(* CoDeSys 2.3.9.28 project: TEST IO.pro *)
(* Libraries: Ethernet.lib 2.12.10 13:48:32, mod_com.lib 2.12.10 13:48:32, ModbusEthernet_04.lib 2.12.10 13:48:36, Standard.lib 2.12.10 13:48:34, SYSLIBCALLBACK.LIB 2.12.10 13:48:32 *)

(* PLC configuration (modules and I/O channels)
0750-0504 4 DO 24V DC 0.5A [Type_10_4_Channels] node 0, in %IB0 out %QB0 {INTTypePAAssignment = PLC; INTTypeModule = plugged}
  AT %QX0.0 [BOOLOnX_Q] Ch_1 Digital output
  AT %QX0.1 [BOOLOnX_Q] Ch_2 Digital output
  AT %QX0.2 [BOOLOnX_Q] Ch_3 Digital output
  AT %QX0.3 [BOOLOnX_Q] Ch_4 Digital output
0750-0403 4 DI 24 V DC 0.2ms [Type_1_4_Channels] node 0, in %IB0 out %QB0 {INTTypePAAssignment = PLC; INTTypeModule = plugged}
  AT %IX0.0 [BOOLOnX_I] Ch_1 Digital input
  AT %IX0.1 [BOOLOnX_I] Ch_2 Digital input
  AT %IX0.2 [BOOLOnX_I] Ch_3 Digital input
  AT %IX0.3 [BOOLOnX_I] Ch_4 Digital input
Fieldbus variables [FB_VARS] node 1, in %IB0 out %QB0
Flag variables [FLAG_VARS] node 2, in %IB0 out %QB0
*)

(* Global variable list: Global_Variables *)
VAR_GLOBAL
	Vystup1: BOOL;
	Vystup2: BOOL;
	Vystup3: BOOL;
	Vystup4: BOOL;
	Vystup5: BOOL;
	Vystup6: BOOL;
	Vystup7: BOOL;
	Vystup8: BOOL;
	Vystup9: BOOL;
	Vystup10: BOOL;
	Vystup11: BOOL;
	Vystup12: BOOL;
	Vystup13: BOOL;
	Vystup14: BOOL;
	Vystup15: BOOL;
	Vystup16: BOOL;
	Vstup1: BOOL;
	Vstup2: BOOL;
	Vstup3: BOOL;
	Vstup4: BOOL;
	Vstup5: BOOL;
	Vstup6: BOOL;
	Vstup7: BOOL;
	Vstup8: BOOL;
	Vstup9: BOOL;
	Vstup10: BOOL;
	Vstup11: BOOL;
	Vstup12: BOOL;
	Vstup13: BOOL;
	Vstup14: BOOL;
	Vstup15: BOOL;
	Vstup16: BOOL;

	Teplota1: WORD;
	Teplota2: WORD;
	Teplota3: WORD;
	Teplota4: WORD;
END_VAR

(* POU PLC_PRG, CFC *)
(*cteni a zapis na vzdalene vstupy/vystupy na SpeedWay DI,DO*)
PROGRAM PLC_PRG
VAR
	Test: SlaveUDP_IO;
	sendStr: ARRAY [1..100] OF WORD;
	RecStr: ARRAY [1..100] OF WORD;
	IPstr:STRING:='192.168.0.201';

	Init: BOOL;
	NoError: BOOL;

	VzdaleneVstupy: WORD_TO_BOOL_16b;
	VydaleneVystupy: BOOL_TO_WORD_16b;
END_VAR
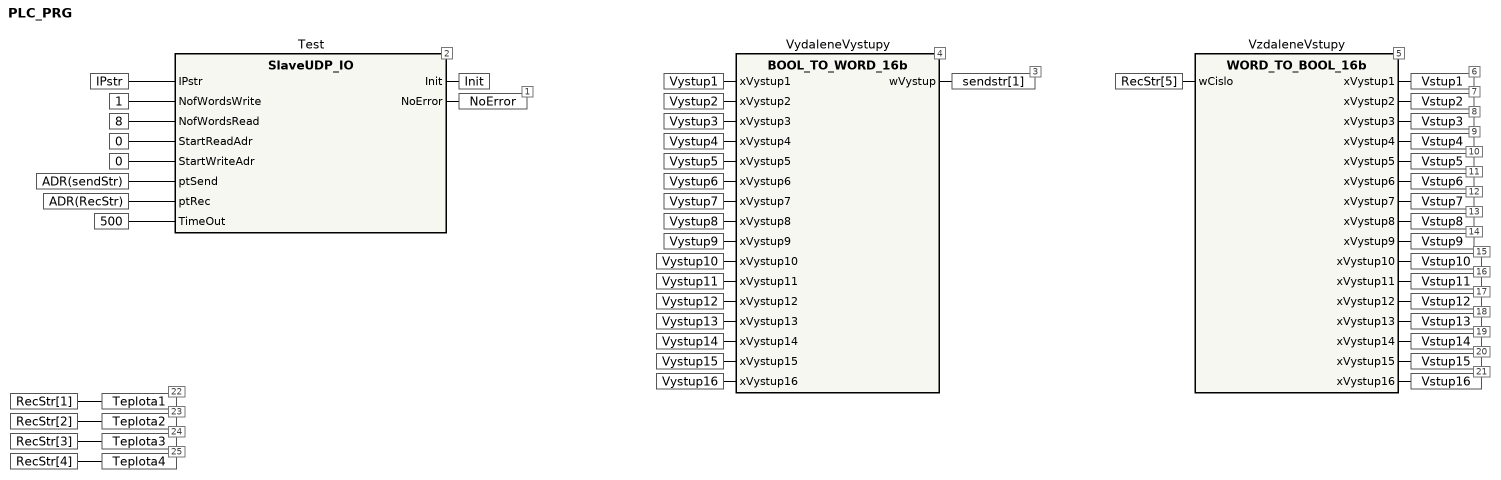
_CFC_ (* Continuous Function Chart, elements in execution order *)
#0 Init <= #2.Init
#1 NoError <= #2.NoError
#2 Test:SlaveUDP_IO(IPstr: IPstr, NofWordsWrite: 1, NofWordsRead: 8, StartReadAdr: 0, StartWriteAdr: 0, ptSend: ADR(sendStr), ptRec: ADR(RecStr), TimeOut: 500)
#3 sendstr[1] <= #4.wVystup
#4 VydaleneVystupy:BOOL_TO_WORD_16b(xVystup1: Vystup1, xVystup2: Vystup2, xVystup3: Vystup3, xVystup4: Vystup4, xVystup5: Vystup5, xVystup6: Vystup6, xVystup7: Vystup7, xVystup8: Vystup8, xVystup9: Vystup9, xVystup10: Vystup10, xVystup11: Vystup11, xVystup12: Vystup12, xVystup13: Vystup13, xVystup14: Vystup14, xVystup15: Vystup15, xVystup16: Vystup16)
#5 VzdaleneVstupy:WORD_TO_BOOL_16b(wCislo: RecStr[5])
#6 Vstup1 <= #5.xVystup1
#7 Vstup2 <= #5.xVystup2
#8 Vstup3 <= #5.xVystup3
#9 Vstup4 <= #5.xVystup4
#10 Vstup5 <= #5.xVystup5
#11 Vstup6 <= #5.xVystup6
#12 Vstup7 <= #5.xVystup7
#13 Vstup8 <= #5.xVystup8
#14 Vstup9 <= #5.xVystup9
#15 Vstup10 <= #5.xVystup10
#16 Vstup11 <= #5.xVystup11
#17 Vstup12 <= #5.xVystup12
#18 Vstup13 <= #5.xVystup13
#19 Vstup14 <= #5.xVystup14
#20 Vstup15 <= #5.xVystup15
#21 Vstup16 <= #5.xVystup16
#22 Teplota1 <= RecStr[1]
#23 Teplota2 <= RecStr[2]
#24 Teplota3 <= RecStr[3]
#25 Teplota4 <= RecStr[4]
_END_CFC_
(* the same logic as Structured Text *)
Init := Test.Init;
NoError := Test.NoError;
Test(IPstr := IPstr, NofWordsWrite := 1, NofWordsRead := 8, StartReadAdr := 0, StartWriteAdr := 0, ptSend := ADR(sendStr), ptRec := ADR(RecStr), TimeOut := 500);
sendstr[1] := VydaleneVystupy.wVystup;
VydaleneVystupy(xVystup1 := Vystup1, xVystup2 := Vystup2, xVystup3 := Vystup3, xVystup4 := Vystup4, xVystup5 := Vystup5, xVystup6 := Vystup6, xVystup7 := Vystup7, xVystup8 := Vystup8, xVystup9 := Vystup9, xVystup10 := Vystup10, xVystup11 := Vystup11, xVystup12 := Vystup12, xVystup13 := Vystup13, xVystup14 := Vystup14, xVystup15 := Vystup15, xVystup16 := Vystup16);
VzdaleneVstupy(wCislo := RecStr[5]);
Vstup1 := VzdaleneVstupy.xVystup1;
Vstup2 := VzdaleneVstupy.xVystup2;
Vstup3 := VzdaleneVstupy.xVystup3;
Vstup4 := VzdaleneVstupy.xVystup4;
Vstup5 := VzdaleneVstupy.xVystup5;
Vstup6 := VzdaleneVstupy.xVystup6;
Vstup7 := VzdaleneVstupy.xVystup7;
Vstup8 := VzdaleneVstupy.xVystup8;
Vstup9 := VzdaleneVstupy.xVystup9;
Vstup10 := VzdaleneVstupy.xVystup10;
Vstup11 := VzdaleneVstupy.xVystup11;
Vstup12 := VzdaleneVstupy.xVystup12;
Vstup13 := VzdaleneVstupy.xVystup13;
Vstup14 := VzdaleneVstupy.xVystup14;
Vstup15 := VzdaleneVstupy.xVystup15;
Vstup16 := VzdaleneVstupy.xVystup16;
Teplota1 := RecStr[1];
Teplota2 := RecStr[2];
Teplota3 := RecStr[3];
Teplota4 := RecStr[4];
END_PROGRAM

(* POU SlaveUDP_IO, ST *)
FUNCTION_BLOCK SlaveUDP_IO
VAR_INPUT
	IPstr:STRING;					(*IP adresa slavu - 750-352,speedwaz etc.*)
	NofWordsWrite:WORD;		(*Pocet wordu, ktere maji byt zapsany*)
	NofWordsRead:WORD;		(*Pocet wordu, tkere maji byt cteny*)
	StartReadAdr:WORD;			(*adresa odkud se bude cist*)
	StartWriteAdr:WORD;			(*odresa kam se bude zapisovat*)
	ptSend:POINTER TO WORD;	(*pointer na pole ktere se bude zapisovat*)
	ptRec:POINTER TO WORD;	(*pointer na pole ktere se bude cist*)
	TimeOut:WORD:=500;		(*cas v milisekundach, pokud neni zadna komunikace, tak potomto case se vystupy nastavi do nuly*)
END_VAR
VAR_OUTPUT
	Init:BOOL;					(*cas do watchdogu byl zapsan a watchdog je spusten -> je mozne komunikovat*)
	NoError:BOOL;			(*zadna chyba pri komunikaci*)
END_VAR
VAR
	state:INT:=0;
	master882: ETHERNET_MODBUSMASTER_UDP;
	start882:BOOL:=FALSE;
	res882:BOOL:=FALSE;
	err882:WORD;
	ready882:BOOL;
	resp882:BYTE;
	ftrig882: F_TRIG;
	tmp_val:WORD;

	ptWrite:POINTER TO BYTE;
	NofWrite:INT;
	WriteAdr:WORD;
END_VAR
IF start882=FALSE THEN
	start882:=TRUE;
	CASE state OF
		0:
			(*zastaveni casovace*)
			tmp_val:=0;
			WriteAdr:=16#100A;
			ptWrite:=ADR(tmp_val);
			NofWrite:=1;
		1:
			(*nastaveni casu, cas je mozne nastavit jen tehdy, kdyz je casovac zastaven*)
			TimeOut:=TimeOut/100;
			tmp_val:=TimeOut;
			NofWordsWrite:=1;
			WriteAdr:=16#1000;
			ptWrite:=ADR(tmp_val);
			NofWrite:=1;
		2:
			(*spusteni watchdogu*)
			tmp_val:=1;
			WriteAdr:=16#100A;
			ptWrite:=ADR(tmp_val);
			NofWrite:=1;
		3:
			(*bezna komunikace*)
			ptWrite:=ptSend;
			NofWrite:=NofWordsWrite;
			WriteAdr:=StartWriteAdr;
	END_CASE;
END_IF;

NofWordsRead;
NofWrite;
IF NofWrite=0 THEN
(*cteni 352 kdyz neni treba nic zapsat*)
master882(strIP_ADDRESS := IPstr,	wPORT := 502,bUNIT_ID := 0,bFUNCTION_CODE := 3,wREAD_ADDRESS := StartReadAdr,wREAD_QUANTITY :=NofWordsRead,
	ptREAD_DATA :=ptRec,wWRITE_ADDRESS := WriteAdr,wWRITE_QUANTITY := NofWrite,ptSEND_DATA :=ptWrite ,xSTART := start882,xRESET := res882,
	tTIME_OUT := t#1s);
ELSE
(*blok pro cteni i zapis v jednom cyklu*)
master882(strIP_ADDRESS := IPstr,	wPORT := 502,bUNIT_ID := 0,bFUNCTION_CODE := 23,wREAD_ADDRESS := StartReadAdr,wREAD_QUANTITY :=NofWordsRead,
	ptREAD_DATA :=ptRec,wWRITE_ADDRESS := WriteAdr,wWRITE_QUANTITY := NofWrite,ptSEND_DATA :=ptWrite ,xSTART := start882,xRESET := res882,
	tTIME_OUT := t#1s);
END_IF;
	(* vystupni promenne *)
	err882:=master882.wERROR;
	ready882:= master882.xREADY;
	resp882:=master882.bRESPONSE_UNIT_ID;

IF master882.wERROR=0 THEN
	NoError:=TRUE;
ELSE
	NoError:=FALSE;
END_IF;
ftrig882(clk:=ready882);
(*prechody ve stavovem automau*)
IF ftrig882.Q   THEN
	 start882:=FALSE;
	IF master882.wERROR=0 THEN
		state:=state+1;	(*neni chyba komunikace, prejdi do dalsiho stavu*)
	ELSE
		IF state>0 AND state<3 THEN
			(*nastala nejaka chyba, vrat so inicializace casovace*)
			state:=0;
		END_IF;
	END_IF;
	IF state>=3 THEN
		state:=3;
		init:=TRUE;
	END_IF;
END_IF;
END_FUNCTION_BLOCK

(* POU Komunikace/WORD_TO_BOOL_16b, ST *)
FUNCTION_BLOCK WORD_TO_BOOL_16b
VAR_INPUT
	wCislo: WORD;

END_VAR
VAR_OUTPUT
	xVystup1: BOOL;
	xVystup2: BOOL;
	xVystup3: BOOL;
	xVystup4: BOOL;
	xVystup5: BOOL;
	xVystup6: BOOL;
	xVystup7: BOOL;
	xVystup8: BOOL;
	xVystup9: BOOL;
	xVystup10: BOOL;
	xVystup11: BOOL;
	xVystup12: BOOL;
	xVystup13: BOOL;
	xVystup14: BOOL;
	xVystup15: BOOL;
	xVystup16: BOOL;
END_VAR
VAR
END_VAR
IF (wCislo > 0)
	THEN
		(*15tı bit*)
		IF(wCislo/32768 > 0)
			THEN
				xVystup16 := TRUE;
				wCislo:= wCislo - 32768;
		ELSE
				xVystup16 := FALSE;
		END_IF

		(*14tı bit*)
		IF(wCislo/16384 > 0)
			THEN
				xVystup15 := TRUE;
				wCislo:= wCislo - 16384;
		ELSE
				xVystup15 := FALSE;
		END_IF

		(*13tı bit*)
		IF(wCislo/8192 > 0)
			THEN
				xVystup14 := TRUE;
				wCislo:= wCislo - 8192;
		ELSE
				xVystup14 := FALSE;
		END_IF

		(*12tı bit*)
		IF(wCislo/4096 > 0)
			THEN
				xVystup13 := TRUE;
				wCislo:= wCislo - 4096;
		ELSE
				xVystup13 := FALSE;
		END_IF

		(*11tı bit*)
		IF(wCislo/2048 > 0)
			THEN
				xVystup12 := TRUE;
				wCislo:= wCislo - 2048;
		ELSE
				xVystup12 := FALSE;
		END_IF

		(*10tı bit*)
		IF(wCislo/1024 > 0)
			THEN
				xVystup11 := TRUE;
				wCislo:= wCislo - 1024;
		ELSE
				xVystup11 := FALSE;
		END_IF

		(*9tı bit*)
		IF(wCislo/512 > 0)
			THEN
				xVystup10 := TRUE;
				wCislo:= wCislo - 512;
		ELSE
				xVystup10 := FALSE;
		END_IF

		(*8tı bit*)
		IF(wCislo/256 > 0)
			THEN
				xVystup9 := TRUE;
				wCislo:= wCislo - 256;
		ELSE
				xVystup9 := FALSE;
		END_IF

		(*7tı bit*)
		IF(wCislo/128 > 0)
			THEN
				xVystup8 := TRUE;
				wCislo:= wCislo - 128;
		ELSE
				xVystup8 := FALSE;
		END_IF

		(*6tı bit*)
		IF(wCislo/64 > 0)
			THEN
				xVystup7 := TRUE;
				wCislo:= wCislo - 64;
		ELSE
				xVystup7 := FALSE;
		END_IF

		(*5tı bit*)
		IF(wCislo/32 > 0)
			THEN
				xVystup6 := TRUE;
				wCislo:= wCislo - 32;
		ELSE
				xVystup6 := FALSE;
		END_IF

		(*4tı bit*)
		IF(wCislo/16 > 0)
			THEN
				xVystup5 := TRUE;
				wCislo:= wCislo - 16;
		ELSE
				xVystup5 := FALSE;
		END_IF

		(*3tí bit*)
		IF(wCislo/8 > 0)
			THEN
				xVystup4 := TRUE;
				wCislo:= wCislo - 8;
		ELSE
				xVystup4 := FALSE;
		END_IF

		(*2hı bit*)
		IF(wCislo/4 > 0)
			THEN
				xVystup3 := TRUE;
				wCislo:= wCislo - 4;
		ELSE
				xVystup3 := FALSE;
		END_IF

		(*1ní bit*)
		IF(wCislo/2 > 0)
			THEN
				xVystup2 := TRUE;
				wCislo:= wCislo - 2;
		ELSE
				xVystup2 := FALSE;
		END_IF

		(*0tı bit*)
		IF(wCislo > 0)
			THEN
				xVystup1 := TRUE;
				wCislo:= wCislo - 1;
		ELSE
				xVystup1 := FALSE;
		END_IF
ELSE
		xVystup1:= FALSE;
		xVystup2:= FALSE;
		xVystup3:= FALSE;
		xVystup4:= FALSE;
		xVystup5:= FALSE;
		xVystup6:= FALSE;
		xVystup7:= FALSE;
		xVystup8:= FALSE;
		xVystup9:= FALSE;
		xVystup10:= FALSE;
		xVystup11:= FALSE;
		xVystup12:= FALSE;
		xVystup13:= FALSE;
		xVystup14:= FALSE;
		xVystup15:= FALSE;
		xVystup16:= FALSE;
END_IF
END_FUNCTION_BLOCK

(* POU Komunikace/BOOL_TO_WORD_16b, CFC *)
FUNCTION_BLOCK BOOL_TO_WORD_16b
VAR_INPUT
	xVystup1: BOOL;
	xVystup2: BOOL;
	xVystup3: BOOL;
	xVystup4: BOOL;
	xVystup5: BOOL;
	xVystup6: BOOL;
	xVystup7: BOOL;
	xVystup8: BOOL;
	xVystup9: BOOL;
	xVystup10: BOOL;
	xVystup11: BOOL;
	xVystup12: BOOL;
	xVystup13: BOOL;
	xVystup14: BOOL;
	xVystup15: BOOL;
	xVystup16: BOOL;
END_VAR
VAR
END_VAR
VAR_OUTPUT
	wVystup: WORD;
END_VAR
VAR (* helpers for the ST form of the networks *)
	_t1 : WORD;
	_t8 : WORD;
	_t11 : WORD;
	_t14 : WORD;
	_t18 : WORD;
	_t21 : WORD;
	_t24 : WORD;
	_t27 : WORD;
	_t30 : WORD;
	_t33 : WORD;
	_t36 : WORD;
	_t39 : WORD;
	_t42 : WORD;
	_t45 : WORD;
	_t48 : WORD;
	_t6 : WORD;
END_VAR
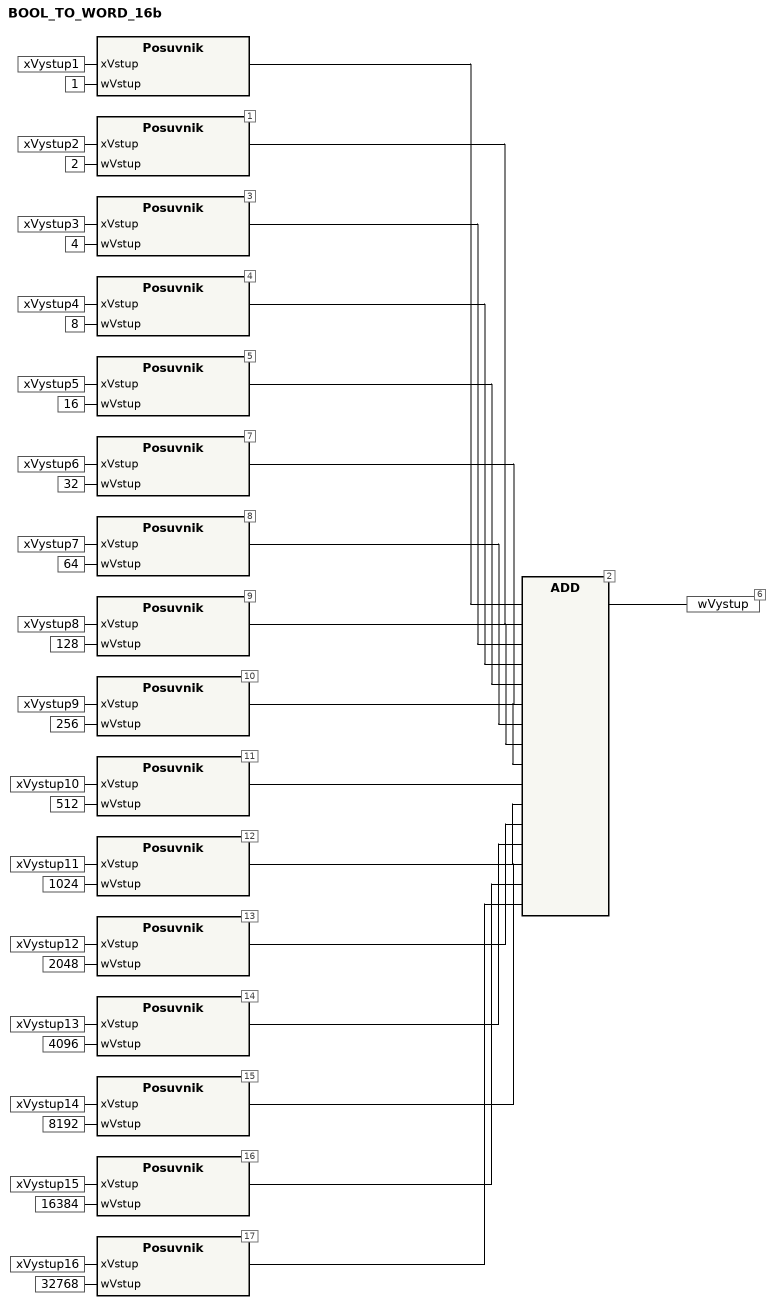
_CFC_ (* Continuous Function Chart, elements in execution order *)
#0 Posuvnik(xVstup: xVystup1, wVstup: 1)
#1 Posuvnik(xVstup: xVystup2, wVstup: 2)
#2 ADD(#0, #1, #3, #4, #5, #7, #8, #9, #10, #11, #12, #13, #14, #15, #16, #17)
#3 Posuvnik(xVstup: xVystup3, wVstup: 4)
#4 Posuvnik(xVstup: xVystup4, wVstup: 8)
#5 Posuvnik(xVstup: xVystup5, wVstup: 16)
#6 wVystup <= #2
#7 Posuvnik(xVstup: xVystup6, wVstup: 32)
#8 Posuvnik(xVstup: xVystup7, wVstup: 64)
#9 Posuvnik(xVstup: xVystup8, wVstup: 128)
#10 Posuvnik(xVstup: xVystup9, wVstup: 256)
#11 Posuvnik(xVstup: xVystup10, wVstup: 512)
#12 Posuvnik(xVstup: xVystup11, wVstup: 1024)
#13 Posuvnik(xVstup: xVystup12, wVstup: 2048)
#14 Posuvnik(xVstup: xVystup13, wVstup: 4096)
#15 Posuvnik(xVstup: xVystup14, wVstup: 8192)
#16 Posuvnik(xVstup: xVystup15, wVstup: 16384)
#17 Posuvnik(xVstup: xVystup16, wVstup: 32768)
_END_CFC_
(* the same logic as Structured Text *)
_t1 := Posuvnik(xVstup := xVystup1, wVstup := 1);
_t6 := _t1 + Posuvnik(xVstup := xVystup2, wVstup := 2) + _t8 + _t11 + _t14 + _t18 + _t21 + _t24 + _t27 + _t30 + _t33 + _t36 + _t39 + _t42 + _t45 + _t48;
_t8 := Posuvnik(xVstup := xVystup3, wVstup := 4);
_t11 := Posuvnik(xVstup := xVystup4, wVstup := 8);
_t14 := Posuvnik(xVstup := xVystup5, wVstup := 16);
wVystup := _t6;
_t18 := Posuvnik(xVstup := xVystup6, wVstup := 32);
_t21 := Posuvnik(xVstup := xVystup7, wVstup := 64);
_t24 := Posuvnik(xVstup := xVystup8, wVstup := 128);
_t27 := Posuvnik(xVstup := xVystup9, wVstup := 256);
_t30 := Posuvnik(xVstup := xVystup10, wVstup := 512);
_t33 := Posuvnik(xVstup := xVystup11, wVstup := 1024);
_t36 := Posuvnik(xVstup := xVystup12, wVstup := 2048);
_t39 := Posuvnik(xVstup := xVystup13, wVstup := 4096);
_t42 := Posuvnik(xVstup := xVystup14, wVstup := 8192);
_t45 := Posuvnik(xVstup := xVystup15, wVstup := 16384);
_t48 := Posuvnik(xVstup := xVystup16, wVstup := 32768);
END_FUNCTION_BLOCK

(* POU Komunikace/Posuvnik, ST *)
FUNCTION Posuvnik : WORD
VAR_INPUT
	xVstup: BOOL;
	wVstup: WORD;
END_VAR
VAR
END_VAR
IF (xVstup = TRUE)
THEN
Posuvnik := wVstup;
ELSE
Posuvnik := 0;
END_IF
END_FUNCTION

(* Visualisation plc_vizu
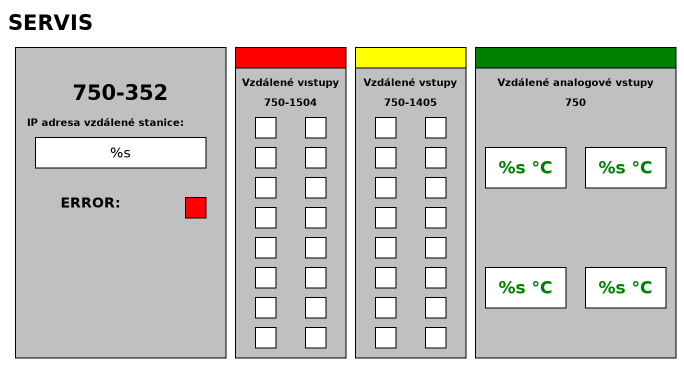
rectangle at (270,120)-(291,141): alarm colour if Vystup1; toggles Vystup1
rectangle at (250,70)-(361,101): text "Vzdálené vıstupy"
rectangle at (320,120)-(341,141): alarm colour if Vystup2; toggles Vystup2
rectangle at (270,150)-(291,171): alarm colour if Vystup3; toggles Vystup3
rectangle at (320,150)-(341,171): alarm colour if Vystup4; toggles Vystup4
rectangle at (270,180)-(291,201): alarm colour if Vystup5; toggles Vystup5
rectangle at (320,180)-(341,201): alarm colour if Vystup6; toggles Vystup6
rectangle at (270,210)-(291,231): alarm colour if Vystup7; toggles Vystup7
rectangle at (320,210)-(341,231): alarm colour if Vystup8; toggles Vystup8
rectangle at (270,240)-(291,261): alarm colour if Vystup9; toggles Vystup9
rectangle at (320,240)-(341,261): alarm colour if Vystup10; toggles Vystup10
rectangle at (270,270)-(291,291): alarm colour if Vystup11; toggles Vystup11
rectangle at (320,270)-(341,291): alarm colour if Vystup12; toggles Vystup12
rectangle at (270,300)-(291,321): alarm colour if Vystup13; toggles Vystup13
rectangle at (320,300)-(341,321): alarm colour if Vystup14; toggles Vystup14
rectangle at (270,330)-(291,351): alarm colour if Vystup15; toggles Vystup15
rectangle at (320,330)-(341,351): alarm colour if Vystup16; toggles Vystup16
rectangle at (10,10)-(121,41): text "SERVIS"
rectangle at (250,90)-(361,121): text "750-1504"
rectangle at (390,120)-(411,141): alarm colour if Vstup1
rectangle at (370,70)-(481,101): text "Vzdálené vstupy"
rectangle at (440,120)-(461,141): alarm colour if Vstup2
rectangle at (390,150)-(411,171): alarm colour if Vstup3
rectangle at (440,150)-(461,171): alarm colour if Vstup4
rectangle at (390,180)-(411,201): alarm colour if Vstup5
rectangle at (440,180)-(461,201): alarm colour if Vstup6
rectangle at (390,210)-(411,231): alarm colour if Vstup7
rectangle at (440,210)-(461,231): alarm colour if Vstup8
rectangle at (390,240)-(411,261): alarm colour if Vstup9
rectangle at (440,240)-(461,261): alarm colour if Vstup10
rectangle at (390,270)-(411,291): alarm colour if Vstup11
rectangle at (440,270)-(461,291): alarm colour if Vstup12
rectangle at (390,300)-(411,321): alarm colour if Vstup13
rectangle at (440,300)-(461,321): alarm colour if Vstup14
rectangle at (390,330)-(411,351): alarm colour if Vstup15
rectangle at (440,330)-(461,351): alarm colour if Vstup16
rectangle at (370,90)-(481,121): text "750-1405"
rectangle at (490,70)-(691,101): text "Vzdálené analogové vstupy"
rectangle at (490,90)-(691,121): text "750"
rounded rectangle at (500,150)-(581,191): text "%s °C"; shows Teplota1/10.0
rounded rectangle at (600,150)-(681,191): text "%s °C"; shows Teplota2/10.0
rounded rectangle at (500,270)-(581,311): text "%s °C"; shows Teplota3/10.0
rounded rectangle at (600,270)-(681,311): text "%s °C"; shows Teplota4/10.0
rectangle at (30,80)-(241,111): text "750-352"
rectangle at (30,110)-(211,141): text "IP adresa vzdálené stanice:"
rectangle at (50,140)-(221,171): text "%s"; shows PLC_PRG.IPstr
rectangle at (200,200)-(221,221): alarm colour if PLC_PRG.NoError
rectangle at (30,190)-(181,221): text "ERROR:"
7 more shapes without text or variables
*)
